PROGRAM Events
VAR
	fbEventosGenerales_PLC:Eventos_PLC;
	bResetArrayAvisos:BOOL;
	bClearEvents:BOOL;
END_VAR

//Eventos Linea 4

fbEventosGenerales_PLC(bClearEvents:=bClearEvents,bResetArrayAvisos:=bResetArrayAvisos);

END_PROGRAM

(* stored: Version 1.1.0.1, ProductVersion 3.1.4024.12
   POU Events: Id {3aea86a1-2655-45e3-a454-ba7e0e35b89c}, SpecialFunc None *)
